GLOBALCONSTANTS AID_IN (* Input number object attribute ids *)
  (* Standard: 61499-1; Description: Copyright (c) 2023 HR Agrartechnik GmbH This program and the accompanying materials are made available under the terms of the Eclipse Public License 2.0 which is available at https://www.eclipse.org/legal/epl-2.0/ SPDX-License-Identifier: EPL-2.0 *)
  (* Version 1.0, 2026-06-20, Franz Höpfinger, HR Agrartechnik GmbH *)
  PACKAGE isobus::UT::Q::const::AID;
  VAR_GLOBAL CONSTANT
    WIDTH : USINT := USINT#1; (* 1: AID_IN_WIDTH - Width in pixels. *)
    HEIGHT : USINT := USINT#2; (* 2: AID_IN_HEIGHT - Height in pixels. *)
    BACKGROUND_COLOUR : USINT := USINT#3; (* 3: AID_IN_BACKGROUND_COLOUR - Background colour index. *)
    FONT_ATT : USINT := USINT#4; (* 4: AID_IN_FONT_ATT - Object ID of a Font Attributes object. *)
    OPTIONS : USINT := USINT#5; (* 5: AID_IN_OPTIONS - Bitmask: Bit 0=Transparent, Bit 1=Display leading zeros, Bit 2=Display zero as blank, Bit 3=Truncate decimals (0=round). *)
    VARIABLE_REF : USINT := USINT#6; (* 6: AID_IN_VARIABLE_REF - Object ID of a Number Variable object. *)
    MIN_VALUE : USINT := USINT#7; (* 7: AID_IN_MIN_VALUE - Minimum value. *)
    MAX_VALUE : USINT := USINT#8; (* 8: AID_IN_MAX_VALUE - Maximum value. *)
    OFFSET : USINT := USINT#9; (* 9: AID_IN_OFFSET - Offset. *)
    SCALE : USINT := USINT#10; (* 10: AID_IN_SCALE - Scale. *)
    NUMB_DECIMALS : USINT := USINT#11; (* 11: AID_IN_NUMB_DECIMALS - Number of decimals. *)
    FORMAT : USINT := USINT#12; (* 12: AID_IN_FORMAT - Format. *)
    JUSTIFICATION : USINT := USINT#13; (* 13: AID_IN_JUSTIFICATION - Justification. *)
    VALUE : USINT := USINT#14; (* 14: AID_IN_VALUE - [14] Read-only for Change Attribute (ISO 11783-6). Query via Get Attribute Value (F.58); update via Change Numeric Value (F.22). *)
    OPTIONS_2 : USINT := USINT#15; (* 15: AID_IN_OPTIONS_2 - [15] Read-only for Change Attribute (ISO 11783-6). Bitmask: Bit 0=Enabled, Bit 1=Real time editing. Query via Get Attribute Value (F.58); manage via Enable/Disable Object (F.4) or Select Input Object (F.6). *)
  END_VAR
END_GLOBALCONSTANTS
